(* CODESYS project SRF08.project

Project tree, tasks and I/O mapping:
  Device : CODESYS Control for Raspberry Pi 64 SL, CODESYS GmbH, order no. 2302000009, version 4.11.0.0
    application Application
      libraries: Standard, 3.5.18.0 (System)
      task MainTask (cyclic, interval t#20ms, priority 1) calls PLC_PRG
      task VISU_TASK (cyclic, interval 100 ms, priority 31) calls VisuElems.Visu_Prg
      program PLC_PRG [ST]
      function block SRF08 [ST]
      visualisation Visualization
      function block Servo [SFC]: LeftStep_active, LeftStep_exit, Power_active, RightStep_active, RightStep_exit
    SoftMotion General Axis Pool
    Camera device
      <Empty>
    GPIOs : GPIOs B+/Pi2, 3S - Smart Software Solutions GmbH, version 4.11.0.0
        unmapped channels: digital inputs (GPIO0..GPIO31), digital outputs (GPIO0..GPIO31)
    I²C
      I2C_master : I2C master, 3S - Smart Software Solutions GmbH, version 4.6.0.0
        Adafruit_PWM_SoftMotion : Adafruit PWM SoftMotion, 3S - Smart Software Solutions GmbH, version 4.11.0.0
          servoDevice : SM_Drive_Servo, 3S - Smart Software Solutions GmbH, version 4.11.0.0
              settings: wDriveID = 0
      I2C_master_1 : I2C master, 3S - Smart Software Solutions GmbH, version 4.11.0.0
    SPI
    Onewire
  text list GlobalTextList
*)

// Device/Application/PLC_PRG
PROGRAM PLC_PRG
VAR
	DistSensor : SRF08 := (_pMaster:= ADR(I2C_Master));
	Servo1 : Servo;
	lrDistance: LREAL;
	lrAccX: LREAL;
	    lrDistance_cm: REAL;     // Distance in centimeters
	    measurementTimer: TON;   // Timer variable
	delayDuration: TIME := T#1S;  // Delay duration (1 second)
	lrMinDistance: LREAL := 0.03;
	
	t: LREAL;
END_VAR

DistSensor();


Servo1();


Servo1.DistanceInput := DistSensor.wBinary;

END_PROGRAM

// Device/Application/SRF08
FUNCTION_BLOCK SRF08 EXTENDS i2c
VAR_INPUT
END_VAR
VAR_OUTPUT
    wBinary : WORD; // Raw distance data from SRF08 in centimeters
END_VAR
VAR
    tDelay          : TON; // Timer for delaying measurement
    tRefreshTime    : TIME := T#200MS; // Time delay for measurement refresh
    bYCommand        : ARRAY[0..1] OF BYTE; // Command bytes to send to the sensor
END_VAR
VAR_TEMP
    highByte, lowByte : BYTE; // Variables to store high and low bytes of the distance data
    udiBytesReceived : DINT; // Number of bytes received from the I2C bus
END_VAR

// Call the parent I2C function block
SUPER^();

CASE _iState OF
    0:
        // Initialize the I2C address for the SRF08 sensor
        usiAddress := 16#70; // Default I2C address for SRF08 sensor
        IF SUPER^.init() THEN
            _iState := 5; // Proceed to the next state after initialization
        END_IF

    5:
        // Set the SRF08 sensor to operate in centimeters mode
        bYCommand[0] := 16#00; // Command register address
        bYCommand[1] := 16#51; // Command to set ranging mode to centimeters
        IF write(ADR(bYCommand), 2) = 2 THEN
            _iState := 10; // Proceed to the next state if the write operation is successful
        END_IF

    10:
        // Wait for a short period before starting the measurement
        tDelay(IN:=TRUE, PT:=tRefreshTime); // Start the delay timer
        IF tDelay.Q THEN
            tDelay(IN:=FALSE); // Stop the delay timer
            bYCommand[0] := 16#02; // Command to initiate measurement
            udiBytesReceived := write(ADR(bYCommand), 1); // Send the measurement command
            _iState := 11; // Proceed to the next state after sending the command
        END_IF

    11:
        // Read the high and low bytes of the distance data
        udiBytesReceived := read(ADR(highByte), 1); // Read the high byte
        IF udiBytesReceived = 1 THEN
            udiBytesReceived := read(ADR(lowByte), 1); // Read the low byte
            IF udiBytesReceived = 1 THEN
                // Combine the high and low bytes into a single WORD
                wBinary := (highByte * 256) + lowByte; // Convert high byte and low byte to distance in centimeters
            END_IF
        END_IF
        _iState := 5; // Prepare for the next measurement cycle

END_CASE

END_FUNCTION_BLOCK

// Device/Application/Servo
FUNCTION_BLOCK Servo
VAR
	lrSpeed: LREAL := 360;
	
	mcp: MC_Power;
	mcma: MC_MoveAbsolute;
	I2C: i2c;
	
	left: BOOL;
	right: BOOL;
	
	wBinary : WORD;

END_VAR

VAR_INPUT
	DistanceInput: WORD;
END_VAR

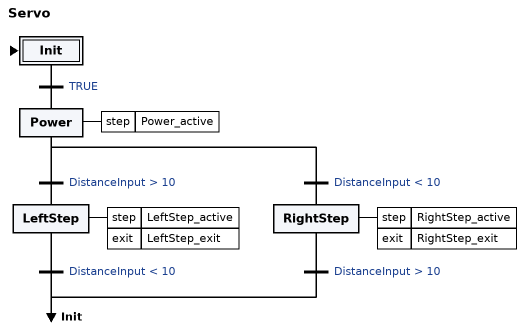
INITIAL_STEP Init:
END_STEP
TRANSITION FROM Init TO Power
    := TRUE;
END_TRANSITION
STEP Power:
    Power_active(N);  // step action
END_STEP
TRANSITION FROM Power TO LeftStep
    := DistanceInput > 10;
END_TRANSITION
STEP LeftStep:
    LeftStep_active(N);  // step action
    LeftStep_exit(P0);  // exit action
END_STEP
TRANSITION FROM LeftStep TO Init
    := DistanceInput < 10;
END_TRANSITION
TRANSITION FROM Power TO RightStep
    := DistanceInput < 10;
END_TRANSITION
STEP RightStep:
    RightStep_active(N);  // step action
    RightStep_exit(P0);  // exit action
END_STEP
TRANSITION FROM RightStep TO Init
    := DistanceInput > 10;
END_TRANSITION

ACTION LeftStep_active:
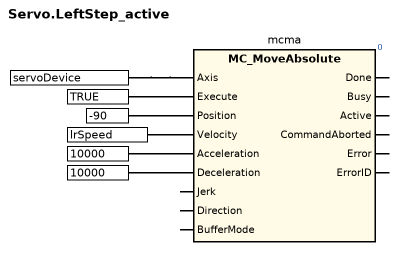
mcma(
    Axis := servoDevice,
    Execute := TRUE,
    Position := -90,
    Velocity := lrSpeed,
    Acceleration := 10000,
    Deceleration := 10000); // MC_MoveAbsolute
END_ACTION

ACTION LeftStep_exit:
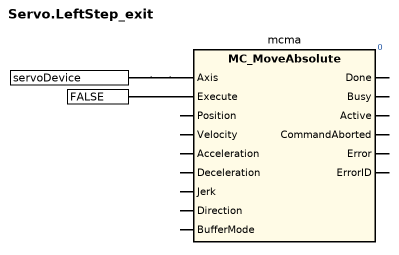
mcma(Axis := servoDevice, Execute := FALSE); // MC_MoveAbsolute
END_ACTION

ACTION Power_active:
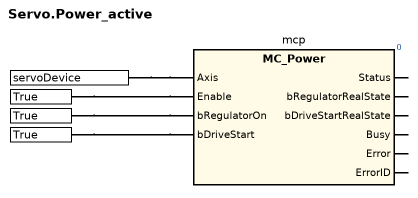
mcp(Axis := servoDevice, Enable := True, bRegulatorOn := True, bDriveStart := True); // MC_Power
END_ACTION

ACTION RightStep_active:
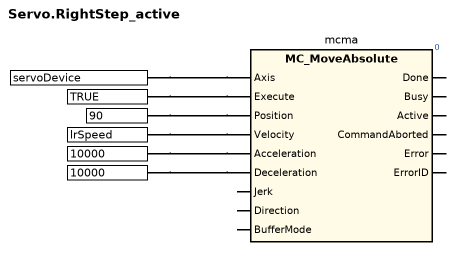
mcma(
    Axis := servoDevice,
    Execute := TRUE,
    Position := 90,
    Velocity := lrSpeed,
    Acceleration := 10000,
    Deceleration := 10000); // MC_MoveAbsolute
END_ACTION

ACTION RightStep_exit:
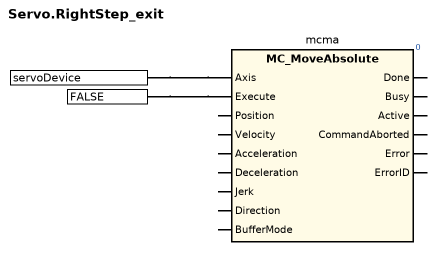
mcma(Axis := servoDevice, Execute := FALSE); // MC_MoveAbsolute
END_ACTION

END_FUNCTION_BLOCK

// Device/Application/Visualization
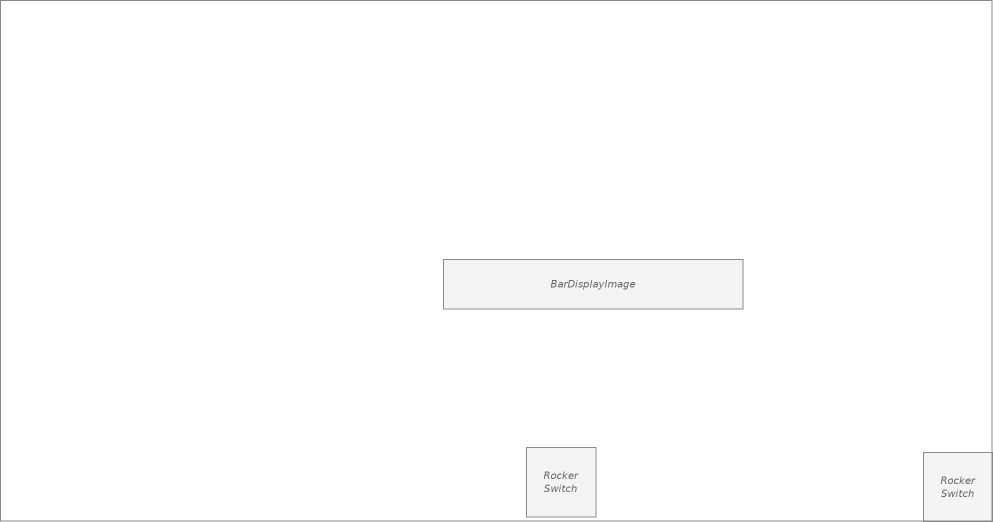
VISUALIZATION Visualization  // 993x522
    BarDisplayImage (443,259 300x50), value: PLC_PRG.DistSensor.wBinary, style: BarDisplayImage-Gray, scale format: %.1f, scale 3..23
    RockerSwitch (923,452 70x70), variable: PLC_PRG.Servo1.right, behaviour: TOGGLE, style: Switch-RockerSwitch-Gray
    RockerSwitch (526,447 70x70), variable: PLC_PRG.Servo1.left, behaviour: TOGGLE, style: Switch-RockerSwitch-Gray
END_VISUALIZATION
